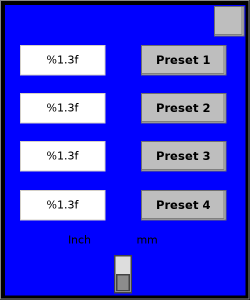
VISUALIZATION Preset_Pellet_Length  // 250x300
    Rectangle (0,0 250x300)
    Textfield (20,45 85x30), "%1.3f", text variable: GVL.Preset1
        OnMouseClick: write the text variable via VisuDialogs.Numpad
    Textfield (20,93 85x30), "%1.3f", text variable: GVL.Preset2
        OnMouseClick: write the text variable via VisuDialogs.Numpad
    Textfield (20,141 85x30), "%1.3f", text variable: GVL.Preset3
        OnMouseClick: write the text variable via VisuDialogs.Numpad
    Textfield (20,190 85x30), "%1.3f", text variable: GVL.Preset4
        OnMouseClick: write the text variable via VisuDialogs.Numpad
    DipSwitch (82,255 82x38), variable: GVL.Metric_Set_Bit, behaviour: TOGGLE, style: Switch-DipSwitch-Gray
    Label (38,225 150x30), "Inch mm"
    Button (141,93 85x30), "Preset 2", text variable: GVL.Preset2
        OnMouseClick: execute {
            IF GVL.Metric_Set_Bit THEN
            	Imperial_Metric_Switching.Pellet_Length_Metric_Input := GVL.Preset2;
            ELSE
            	Imperial_Metric_Switching.Pellet_Length_Imperial_Input := GVL.Preset2;
            END_IF
        }
    Button (141,45 85x30), "Preset 1"
        OnMouseClick: execute {
            IF GVL.Metric_Set_Bit THEN
            	Imperial_Metric_Switching.Pellet_Length_Metric_Input := GVL.Preset1;
            ELSE
            	Imperial_Metric_Switching.Pellet_Length_Imperial_Input := GVL.Preset1;
            END_IF
        }
    Button (141,141 85x30), "Preset 3", text variable: GVL.Preset3
        OnMouseClick: execute {
            IF GVL.Metric_Set_Bit THEN
            	Imperial_Metric_Switching.Pellet_Length_Metric_Input := GVL.Preset3;
            ELSE
            	Imperial_Metric_Switching.Pellet_Length_Imperial_Input := GVL.Preset3;
            END_IF
        }
    Button (141,190 85x30), "Preset 4", text variable: GVL.Preset4
        OnMouseClick: execute {
            IF GVL.Metric_Set_Bit THEN
            	Imperial_Metric_Switching.Pellet_Length_Metric_Input := GVL.Preset4;
            ELSE
            	Imperial_Metric_Switching.Pellet_Length_Imperial_Input := GVL.Preset4;
            END_IF
        }
    Button (214,6 30x30), image: VisuSymbols.Symbols.Wrong
        OnMouseClick: CloseDialog Dialog=Preset_Pellet_Length, Result=None, NumpadKeypadSet=True
END_VISUALIZATION

(* stored: Version 1.1.0.1, ProductVersion 3.1.4024.12
   Visu Preset_Pellet_Length: Id {0932efbd-38c4-4883-b64f-1c4e0e2e5dba} *)
